# EPICS autosave request: lsredis/iocBoot/iocvxWorks/auto_settings.req
# Note: the macro P must have been supplied to the routine that parses
# this file.  Normally, this means a command like the following will be issued
# after iocInit:
# create_monitor_set("auto_settings.req",30,"P=lsredis:")

file built_settings.req P=$(P)
